// ============================================================================
// FB_1001_Station1.scl - 汇川换型改造 工位1 动作机构控制功能块
// ============================================================================
// 描述:
//   实现 DJ-2026-009 汇川换型改造 工位1 进料、定位、夹紧、加工与出料控制.
//   严格遵循 LSP-905 语法白名单、DINT 毫秒定时器三段式、CASE 防死锁 ELSE 与结构体整块传递.
//   遵循 STD-840 设备抽象, STD-820 8步握手.
// ============================================================================

FUNCTION_BLOCK FB_1001_Station1

VAR_IN_OUT
    io_stStation    : ST_Station1;      // 工位1 全局交互结构体 (整块传递)
    io_stExternal   : ST_ExternalDevice;// 外部设备 8步握手交握结构体
END_VAR

VAR
    // 局部状态变量
    s_iStep         : DINT;             // 内部工步号
    s_bRunning      : BOOL;             // 运行中状态
    s_bDone         : BOOL;             // 本周期完成脉冲
    s_bAlarm        : BOOL;             // 站级报警
    s_iAlarmCode    : DINT;             // 报警代码

    // 定时器实例 (DINT 毫秒三段式, 遵循 LSP-906/903)
    s_tStepTimer    : FB_TON;           // 工步计时器 (ms)
    s_tProcessTimer : FB_TON;           // 工艺加工计时器 (ms)
END_VAR

VAR_TEMP
    t_bAutoEnable   : BOOL;
    t_bReset        : BOOL;
    t_bInPos        : BOOL;
    t_bWorkPos      : BOOL;
    t_dCylTimeout   : DINT;
    t_dProcessTime  : DINT;
END_VAR

CONST
    STEP_IDLE           : DINT := 0;    // 待机就绪
    STEP_WAIT_MATERIAL  : DINT := 1;    // 等待来料 (STD-820)
    STEP_FEEDING        : DINT := 2;    // 进料输送
    STEP_CLAMP          : DINT := 10;   // 夹紧顶升
    STEP_PROCESS        : DINT := 20;   // 工艺加工
    STEP_RELEASE_UNLOAD : DINT := 30;   // 松开出料
    STEP_FAULT          : DINT := 99;   // 故障保护
END_CONST

BEGIN
    // =========================================================================
    // 0. 定时器顶部批量无条件调用 (LSP-906/903)
    // =========================================================================
    s_tStepTimer(IN := s_tStepTimer.IN, PT := s_tStepTimer.PT, Q => s_tStepTimer.Q, ET => s_tStepTimer.ET);
    s_tProcessTimer(IN := s_tProcessTimer.IN, PT := s_tProcessTimer.PT, Q => s_tProcessTimer.Q, ET => s_tProcessTimer.ET);

    // =========================================================================
    // 1. 解包临时变量
    // =========================================================================
    t_bAutoEnable  := io_stStation.stControl.bAutoEnable;
    t_bReset       := io_stStation.stControl.bReset;
    t_bInPos       := io_stStation.stSensors.bInPosSensor;
    t_bWorkPos     := io_stStation.stSensors.bWorkPosSensor;

    t_dCylTimeout  := io_stStation.stConfig.dCylTimeoutMs;
    IF t_dCylTimeout <= 0 THEN
        t_dCylTimeout := 5000; // 默认 5000ms
    END_IF;

    t_dProcessTime := io_stStation.stConfig.dProcessTimeMs;
    IF t_dProcessTime <= 0 THEN
        t_dProcessTime := 2000; // 默认 2000ms
    END_IF;

    // =========================================================================
    // 2. 故障复位
    // =========================================================================
    IF t_bReset THEN
        s_bAlarm := FALSE;
        s_iAlarmCode := 0;
        IF s_iStep = STEP_FAULT OR (s_iStep <> STEP_IDLE AND NOT t_bAutoEnable) THEN
            s_iStep := STEP_IDLE;
        END_IF;
    END_IF;

    // =========================================================================
    // 3. 主工步状态机
    // =========================================================================
    IF NOT t_bAutoEnable OR s_bAlarm THEN
        // 非使能或报警模式下，安全保持，撤销所有设备命令
        io_stStation.stActuators.stMotorFwd.i_bFwdReq := FALSE;
        io_stStation.stActuators.stCyl1.stCmd.Extend := FALSE;
        io_stStation.stActuators.stCyl1.stCmd.Retract := TRUE;
        io_stStation.stActuators.stCyl2.stCmd.Extend := FALSE;
        io_stStation.stActuators.stCyl2.stCmd.Retract := TRUE;

        // 撤销握手准备信号
        io_stExternal.stUpstream.bMachine_ReadyIn := FALSE;
        io_stExternal.stDownstream.bMachine_ReadyOut := FALSE;

        s_bRunning := FALSE;
        s_bDone := FALSE;
        s_tStepTimer.IN := FALSE;
        s_tProcessTimer.IN := FALSE;

        IF s_bAlarm THEN
            s_iStep := STEP_FAULT;
        ELSE
            s_iStep := STEP_IDLE;
        END_IF;
    ELSE
        s_bRunning := TRUE;

        CASE s_iStep OF
            STEP_IDLE:
                s_bDone := FALSE;
                io_stStation.stActuators.stMotorFwd.i_bFwdReq := FALSE;
                io_stStation.stActuators.stCyl1.stCmd.Extend := FALSE;
                io_stStation.stActuators.stCyl1.stCmd.Retract := TRUE;
                io_stStation.stActuators.stCyl2.stCmd.Extend := FALSE;
                io_stStation.stActuators.stCyl2.stCmd.Retract := TRUE;

                // 配置气缸超时参数
                io_stStation.stActuators.stCyl1.stCmd.TimeoutMs := t_dCylTimeout;
                io_stStation.stActuators.stCyl2.stCmd.TimeoutMs := t_dCylTimeout;

                // 等待气缸回原点
                IF io_stStation.stActuators.stCyl1.stSts.IsRetracted AND io_stStation.stActuators.stCyl2.stSts.IsRetracted THEN
                    s_iStep := STEP_WAIT_MATERIAL;
                    s_tStepTimer.IN := FALSE;
                END_IF;

            STEP_WAIT_MATERIAL:
                // 发出准备好信号，由 FB_3001 负责上游交握
                io_stExternal.stUpstream.bMachine_ReadyIn := TRUE;

                // 等待 FB_3001 状态机推进至允许进料或收到进料请求
                // 根据 STD-820，FB_3001 的 iInfeedStep >= 30 表示允许电机动作
                IF io_stExternal.stUpstream.iInfeedStep >= 30 THEN
                    s_iStep := STEP_FEEDING;
                    s_tStepTimer.IN := FALSE;
                    io_stExternal.stUpstream.bMachine_ReadyIn := FALSE; // 撤销就绪
                END_IF;

            STEP_FEEDING:
                io_stStation.stActuators.stMotorFwd.i_bFwdReq := TRUE;

                s_tStepTimer.IN := TRUE;
                s_tStepTimer.PT := 10000; // 进料超时 10s

                IF t_bWorkPos THEN
                    io_stStation.stActuators.stMotorFwd.i_bFwdReq := FALSE;
                    s_iStep := STEP_CLAMP;
                    s_tStepTimer.IN := FALSE;
                ELSIF s_tStepTimer.Q THEN
                    s_bAlarm := TRUE;
                    s_iAlarmCode := 101; // 进料超时报警
                    io_stStation.stActuators.stMotorFwd.i_bFwdReq := FALSE;
                    s_iStep := STEP_FAULT;
                END_IF;

            STEP_CLAMP:
                io_stStation.stActuators.stCyl1.stCmd.Extend := TRUE;
                io_stStation.stActuators.stCyl1.stCmd.Retract := FALSE;
                io_stStation.stActuators.stCyl2.stCmd.Extend := TRUE;
                io_stStation.stActuators.stCyl2.stCmd.Retract := FALSE;

                // STD-840: 等待状态输入
                IF io_stStation.stActuators.stCyl1.stSts.IsExtended AND io_stStation.stActuators.stCyl2.stSts.IsExtended THEN
                    s_iStep := STEP_PROCESS;
                    s_tStepTimer.IN := FALSE;
                ELSIF io_stStation.stActuators.stCyl1.stSts.Timeout OR io_stStation.stActuators.stCyl2.stSts.Timeout THEN
                    s_bAlarm := TRUE;
                    s_iAlarmCode := 102; // 夹紧/顶升超时报警
                    s_iStep := STEP_FAULT;
                END_IF;

            STEP_PROCESS:
                // 启动工艺加工定时器
                s_tProcessTimer.IN := TRUE;
                s_tProcessTimer.PT := t_dProcessTime;

                IF s_tProcessTimer.Q THEN
                    s_iStep := STEP_RELEASE_UNLOAD;
                    s_tProcessTimer.IN := FALSE;
                    s_tStepTimer.IN := FALSE;
                END_IF;

            STEP_RELEASE_UNLOAD:
                io_stStation.stActuators.stCyl1.stCmd.Extend := FALSE;
                io_stStation.stActuators.stCyl1.stCmd.Retract := TRUE;
                io_stStation.stActuators.stCyl2.stCmd.Extend := FALSE;
                io_stStation.stActuators.stCyl2.stCmd.Retract := TRUE;

                IF io_stStation.stActuators.stCyl1.stSts.IsRetracted AND io_stStation.stActuators.stCyl2.stSts.IsRetracted THEN
                    io_stStation.stActuators.stMotorFwd.i_bFwdReq := TRUE;

                    s_tStepTimer.IN := TRUE;
                    s_tStepTimer.PT := 10000; // 出料超时 10s

                    // STD-820 出料握手：等待下游交握完成 (iOutfeedStep 走完) 且工件离开本站
                    // FB_3001 负责与下游交握，本站主要监测工件离开
                    io_stExternal.stDownstream.bMachine_ReadyOut := TRUE;

                    IF NOT t_bWorkPos AND NOT t_bInPos THEN
                        io_stStation.stActuators.stMotorFwd.i_bFwdReq := FALSE;
                        s_bDone := TRUE;
                        s_iStep := STEP_IDLE;
                        s_tStepTimer.IN := FALSE;
                        io_stExternal.stDownstream.bMachine_ReadyOut := FALSE;
                    ELSIF s_tStepTimer.Q THEN
                        s_bAlarm := TRUE;
                        s_iAlarmCode := 103; // 松开/出料超时报警
                        io_stStation.stActuators.stMotorFwd.i_bFwdReq := FALSE;
                        s_iStep := STEP_FAULT;
                    END_IF;
                ELSIF io_stStation.stActuators.stCyl1.stSts.Timeout OR io_stStation.stActuators.stCyl2.stSts.Timeout THEN
                    s_bAlarm := TRUE;
                    s_iAlarmCode := 104; // 缩回超时报警
                    s_iStep := STEP_FAULT;
                END_IF;

            STEP_FAULT:
                s_bRunning := FALSE;
                s_tStepTimer.IN := FALSE;
                s_tProcessTimer.IN := FALSE;

            ELSE
                // 防死锁安全分支
                s_iStep := STEP_IDLE;
                s_tStepTimer.IN := FALSE;
                s_tProcessTimer.IN := FALSE;
        END_CASE;
    END_IF;

    // =========================================================================
    // 4. 统一末尾封包与回写
    // =========================================================================
    io_stStation.stStatus.iStep       := s_iStep;
    io_stStation.stStatus.bRunning     := s_bRunning;
    io_stStation.stStatus.bDone        := s_bDone;
    io_stStation.stStatus.bAlarm       := s_bAlarm;
    io_stStation.stStatus.iAlarmCode   := s_iAlarmCode;
    io_stStation.stStatus.bWaitMaterial:= (s_iStep = STEP_WAIT_MATERIAL);
    io_stStation.stStatus.bProcessing  := (s_iStep = STEP_PROCESS);

END_FUNCTION_BLOCK
